SYSTEM TestEDELAY (* System Configuration *)
  (* Standard: 61499-1 *)
  (* Version 0.3, 2003-12-05, JHC, Rockwell Automation, Renamed from NEWSYSTEM. *)
  (* Version 0.2, 2002-11-05, JHC, Rockwell Automation, Fixed missing (empty) FBD in Application. *)
  (* Version 0.1, 2002-01-17, JHC, Rockwell Automation, Minor cleanup *)
  (* Version 0.0, 2000-05-27, JHC, Rockwell Automation *)
  APPLICATION APP1
  END_APPLICATION
  DEVICE DEV1 : FRAME_DEVICE(BOUNDS := [0,0,100,100])
    RESOURCE RES1 : PANEL_RESOURCE
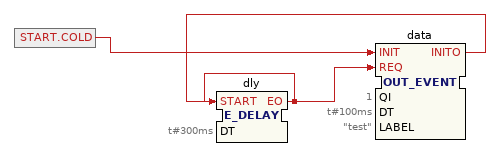
      FBS
        data : OUT_EVENT(QI := 1, DT := t#100ms, LABEL := "test");
        dly : E_DELAY(DT := t#300ms);
      END_FBS
      EVENT_CONNECTIONS
        START.COLD TO data.INIT;
        data.INITO TO dly.START;
        dly.EO TO dly.START;
        dly.EO TO data.REQ;
      END_CONNECTIONS
    END_RESOURCE
  END_DEVICE
END_SYSTEM
